// TIA Portal V20 export
TYPE "LER_typeBrakeTestEmPlcCommands"
// stored: Access Published
   STRUCT
      brakeSelect : Bool;
      brakeStart : Bool;
      axisReset : Bool;
   END_STRUCT;
END_TYPE
